// TIA Portal V20 export
FUNCTION_BLOCK "LER_EQP_m_Communication"   // FB221, LAD
// stored: Access Published, MemoryReserve 100, SetENOAutomatically false
   VAR_INPUT
      Enable : Bool;
      RcvHearBeat : Byte;
   END_VAR
   VAR_OUTPUT
      error : Bool;
      status : Word;
   END_VAR
   VAR_IN_OUT
      CommunicationSEND : Variant;
      CommunicationRCV : Variant;
      configuration : "LER_typeCommunicationConfiguration";
      moduleInterface : "LER_typeCommunicationInterface";
      controlNode : "LER_typeCommunicationControlNode";
   END_VAR
   VAR
      instBSEND { S7_SetPoint := 'True'} : BSEND;
      instBRCV { S7_SetPoint := 'True'} : BRCV;
      statBSEND : "LER_typeCommunicationBSENDParameter";
      statBRCV { S7_SetPoint := 'True'} : "LER_typeCommunicationBRCVParameter";
      statTonTimer : Array[0..9] of TON_TIME;
      statHeartBeat { S7_SetPoint := 'True'} : Byte;
      statDisableAlarms : Bool;
   END_VAR
   VAR CONSTANT
      STATUS_NO_ERROR_OCCURRED : Word := 16#0;
      ERR_COMMUNICATION_ERROR : Word := 16#8000;
   END_VAR
BEGIN

REGION Network 1 (SCL): ##### Inputs mapping #####
   #statDisableAlarms := #configuration.disableAlarms;
   #statBRCV.Input.EN_R := TRUE;
END_REGION

REGION Network 2: BSEND REQUEST
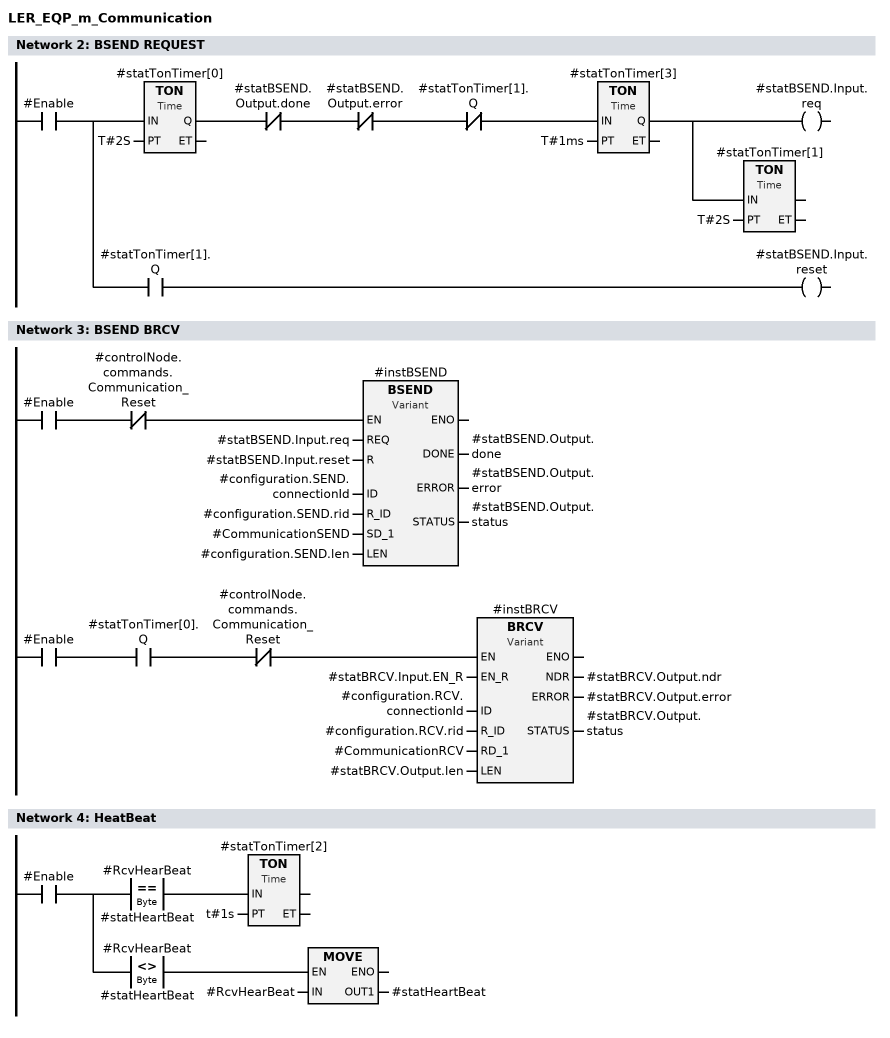
   RUNG wire#powerrail
      Contact( #Enable )
      wire#w1
      { S7_Templates := "time_type := Time" } #statTonTimer[0].TON(pt := T#2S, et =>)
      I_Contact( #statBSEND.Output.done )
      I_Contact( #statBSEND.Output.error )
      I_Contact( #statTonTimer[1].Q )
      { S7_Templates := "time_type := Time" } #statTonTimer[3].TON(pt := T#1ms, et =>)
      wire#w2
      Coil( #statBSEND.Input.req )
   END_RUNG
   RUNG wire#w2
      { S7_Templates := "time_type := Time" } #statTonTimer[1].TON(pt := T#2S, et =>)
   END_RUNG
   RUNG wire#w1
      Contact( #statTonTimer[1].Q )
      Coil( #statBSEND.Input.reset )
   END_RUNG
   // the same network as SCL:
   #statTonTimer[0].TON(IN := #Enable, PT := T#2S);
   #statTonTimer[3].TON(IN := #statTonTimer[0].Q AND NOT #statBSEND.Output.done AND NOT #statBSEND.Output.error AND NOT #statTonTimer[1].Q,
                        PT := T#1ms);
   #statBSEND.Input.req := #statTonTimer[3].Q;
   #statTonTimer[1].TON(IN := #statTonTimer[3].Q, PT := T#2S);
   #statBSEND.Input.reset := #Enable AND #statTonTimer[1].Q;
END_REGION

REGION Network 3: BSEND BRCV
   RUNG wire#powerrail
      Contact( #Enable )
      I_Contact( #controlNode.commands.Communication_Reset )
      { S7_Templates := "[ptr_type := Variant, id_type := CONN_PRG, r_id_type := CONN_R_ID]" } #instBSEND.BSEND(REQ := #statBSEND.Input.req, R := #statBSEND.Input.reset, ID := #configuration.SEND.connectionId, R_ID := #configuration.SEND.rid, SD_1 := #CommunicationSEND, LEN := #configuration.SEND.len, DONE => #statBSEND.Output.done, ERROR => #statBSEND.Output.error, STATUS => #statBSEND.Output.status)
   END_RUNG
   RUNG wire#powerrail
      Contact( #Enable )
      Contact( #statTonTimer[0].Q )
      I_Contact( #controlNode.commands.Communication_Reset )
      { S7_Templates := "[ptr_type := Variant, id_type := CONN_PRG, r_id_type := CONN_R_ID]" } #instBRCV.BRCV(EN_R := #statBRCV.Input.EN_R, ID := #configuration.RCV.connectionId, R_ID := #configuration.RCV.rid, RD_1 := #CommunicationRCV, LEN := #statBRCV.Output.len, NDR => #statBRCV.Output.ndr, ERROR => #statBRCV.Output.error, STATUS => #statBRCV.Output.status)
   END_RUNG
   // the same network as SCL:
   IF #Enable AND NOT #controlNode.commands.Communication_Reset THEN
       #instBSEND(REQ := #statBSEND.Input.req,   // BSEND
                  R := #statBSEND.Input.reset,
                  ID := #configuration.SEND.connectionId,
                  R_ID := #configuration.SEND.rid,
                  SD_1 := #CommunicationSEND,
                  LEN := #configuration.SEND.len,
                  DONE => #statBSEND.Output.done,
                  ERROR => #statBSEND.Output.error,
                  STATUS => #statBSEND.Output.status);
   END_IF;
   IF #Enable AND #statTonTimer[0].Q AND NOT #controlNode.commands.Communication_Reset THEN
       #instBRCV(EN_R := #statBRCV.Input.EN_R,   // BRCV
                 ID := #configuration.RCV.connectionId,
                 R_ID := #configuration.RCV.rid,
                 RD_1 := #CommunicationRCV,
                 LEN := #statBRCV.Output.len,
                 NDR => #statBRCV.Output.ndr,
                 ERROR => #statBRCV.Output.error,
                 STATUS => #statBRCV.Output.status);
   END_IF;
END_REGION

REGION Network 4: HeatBeat
   RUNG wire#powerrail
      Contact( #Enable )
      wire#w1
      { S7_Templates := "SrcType := Byte" } EQ_Contact(in1 := #RcvHearBeat, in2 := #statHeartBeat)
      { S7_Templates := "time_type := Time" } #statTonTimer[2].TON(pt := t#1s, et =>)
   END_RUNG
   RUNG wire#w1
      { S7_Templates := "SrcType := Byte" } NE_Contact(in1 := #RcvHearBeat, in2 := #statHeartBeat)
      Move(in := #RcvHearBeat, out1 => #statHeartBeat)
   END_RUNG
   // the same network as SCL:
   #statTonTimer[2].TON(IN := #Enable AND (#RcvHearBeat = #statHeartBeat), PT := t#1s);
   IF #Enable AND (#RcvHearBeat <> #statHeartBeat) THEN #statHeartBeat := #RcvHearBeat; END_IF;
END_REGION

REGION Network 5 (SCL): Error Check
   REGION  Error Code Search

       IF #Enable THEN    // Hardwere ID mapping Error
           IF #statBSEND.Output.error THEN
               #status := #statBSEND.Output.status;

           ELSIF #statBRCV.Output.error THEN
               #status := #statBRCV.Output.status;

           ELSIF #statTonTimer[2].Q THEN
               #status := #ERR_COMMUNICATION_ERROR;

           ELSE
               #status := #STATUS_NO_ERROR_OCCURRED;

           END_IF;
       ELSE
           #error := FALSE;
           #status := #STATUS_NO_ERROR_OCCURRED;

       END_IF;


   END_REGION


   // Error Bit
   #error := #status <> 0;
END_REGION

REGION Network 6 (SCL): ##### Outputs mapping #####
   #moduleInterface.monitoring.error := #error;
   #moduleInterface.monitoring.status := #status;

   #controlNode.monitoring := #moduleInterface.monitoring;
END_REGION
END_FUNCTION_BLOCK
